FUNCTION_BLOCK CVCAMERA (* Camera OpenCV function block *)
  (* Version 1.0, AN, SWDC RTSoft *)
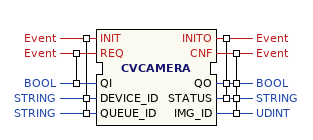
  EVENT_INPUT
    INIT WITH DEVICE_ID, QUEUE_ID;
    REQ WITH QI;
  END_EVENT
  EVENT_OUTPUT
    INITO WITH QO, STATUS;
    CNF WITH QO, IMG_ID, STATUS;
  END_EVENT
  VAR_INPUT
    QI : BOOL;
    DEVICE_ID : STRING;
    QUEUE_ID : STRING;
  END_VAR
  VAR_OUTPUT
    QO : BOOL;
    STATUS : STRING;
    IMG_ID : UDINT;
  END_VAR
  (* Service APPLICATION/RESOURCE: Service Interface Function Block Type *)
END_FUNCTION_BLOCK
